SYSTEM CODEC_TESTL (* PUBL/SUBL Test *)
  (* Standard: 61499 Feasibility Demo *)
  (* Version 0.0, 2001-10-04, JHC, Rockwell Automation, Copied/modified from CODEC_TEST *)
  APPLICATION TEST_BITS (* Test bit string data types *)
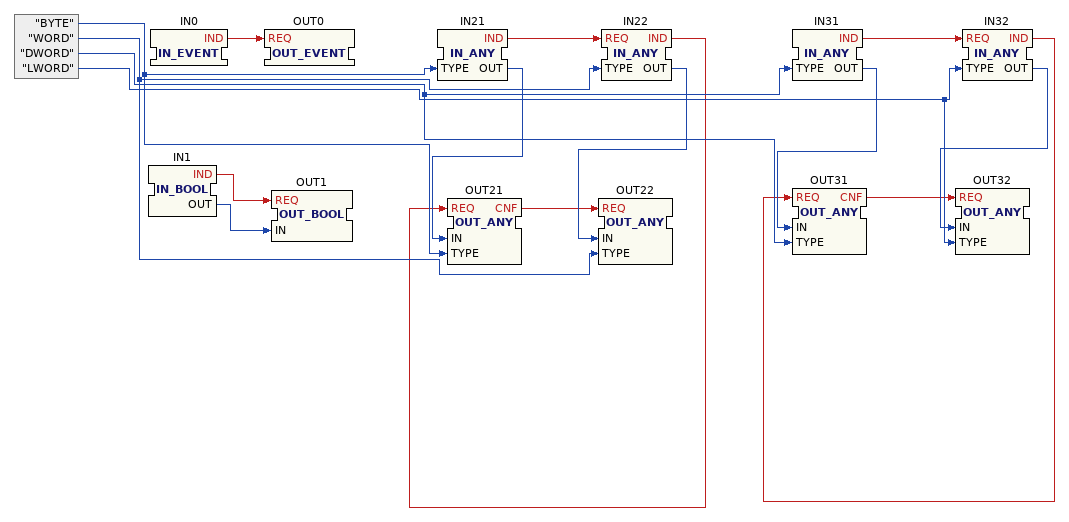
    FBS
      IN0 : IN_EVENT;
      OUT0 : OUT_EVENT;
      IN1 : IN_BOOL;
      OUT1 : OUT_BOOL;
      IN21 : IN_ANY;
      OUT21 : OUT_ANY;
      IN22 : IN_ANY;
      OUT22 : OUT_ANY;
      IN31 : IN_ANY;
      OUT31 : OUT_ANY;
      IN32 : IN_ANY;
      OUT32 : OUT_ANY;
    END_FBS
    EVENT_CONNECTIONS
      IN0.IND TO OUT0.REQ;
      IN1.IND TO OUT1.REQ;
      IN21.IND TO IN22.REQ;
      IN22.IND TO OUT21.REQ;
      OUT21.CNF TO OUT22.REQ;
      IN31.IND TO IN32.REQ;
      IN32.IND TO OUT31.REQ;
      OUT31.CNF TO OUT32.REQ;
    END_CONNECTIONS
    DATA_CONNECTIONS
      IN1.OUT TO OUT1.IN;
      IN21.OUT TO OUT21.IN;
      IN22.OUT TO OUT22.IN;
      IN31.OUT TO OUT31.IN;
      IN32.OUT TO OUT32.IN;
      "BYTE" TO IN21.TYPE;
      "BYTE" TO OUT21.TYPE;
      "WORD" TO IN22.TYPE;
      "WORD" TO OUT22.TYPE;
      "DWORD" TO IN31.TYPE;
      "DWORD" TO OUT31.TYPE;
      "LWORD" TO IN32.TYPE;
      "LWORD" TO OUT32.TYPE;
    END_CONNECTIONS
  END_APPLICATION
  APPLICATION TEST_INTS (* Test integer data types *)
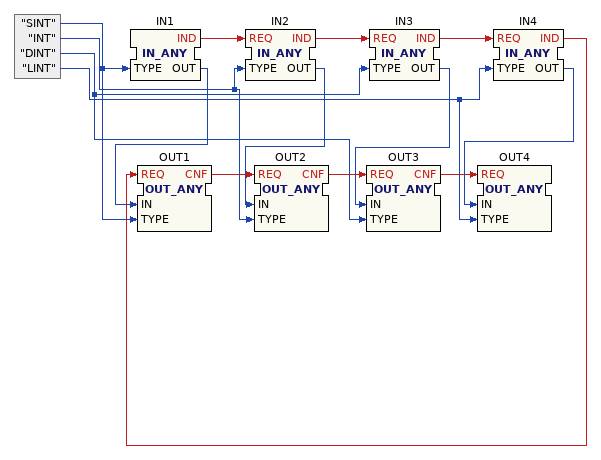
    FBS
      IN1 : IN_ANY;
      IN2 : IN_ANY;
      IN3 : IN_ANY;
      IN4 : IN_ANY;
      OUT1 : OUT_ANY;
      OUT2 : OUT_ANY;
      OUT3 : OUT_ANY;
      OUT4 : OUT_ANY;
    END_FBS
    EVENT_CONNECTIONS
      IN1.IND TO IN2.REQ;
      IN2.IND TO IN3.REQ;
      IN3.IND TO IN4.REQ;
      IN4.IND TO OUT1.REQ;
      OUT1.CNF TO OUT2.REQ;
      OUT2.CNF TO OUT3.REQ;
      OUT3.CNF TO OUT4.REQ;
    END_CONNECTIONS
    DATA_CONNECTIONS
      IN1.OUT TO OUT1.IN;
      IN2.OUT TO OUT2.IN;
      IN3.OUT TO OUT3.IN;
      IN4.OUT TO OUT4.IN;
      "SINT" TO IN1.TYPE;
      "SINT" TO OUT1.TYPE;
      "INT" TO IN2.TYPE;
      "INT" TO OUT2.TYPE;
      "DINT" TO IN3.TYPE;
      "DINT" TO OUT3.TYPE;
      "LINT" TO IN4.TYPE;
      "LINT" TO OUT4.TYPE;
    END_CONNECTIONS
  END_APPLICATION
  APPLICATION TEST_UINTS (* Test unsigned integer data types *)
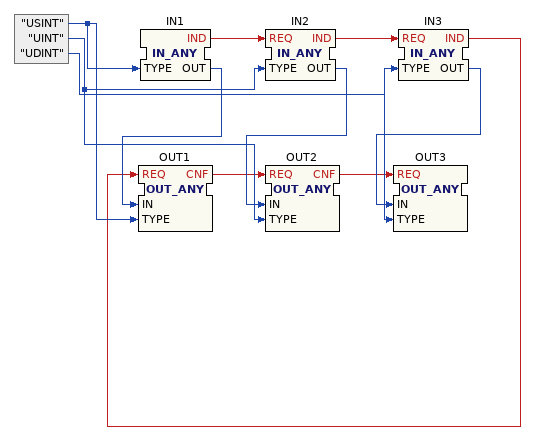
    FBS
      IN1 : IN_ANY;
      IN2 : IN_ANY;
      IN3 : IN_ANY;
      OUT1 : OUT_ANY;
      OUT2 : OUT_ANY;
      OUT3 : OUT_ANY;
    END_FBS
    EVENT_CONNECTIONS
      IN1.IND TO IN2.REQ;
      IN2.IND TO IN3.REQ;
      IN3.IND TO OUT1.REQ;
      OUT1.CNF TO OUT2.REQ;
      OUT2.CNF TO OUT3.REQ;
    END_CONNECTIONS
    DATA_CONNECTIONS
      IN1.OUT TO OUT1.IN;
      IN2.OUT TO OUT2.IN;
      IN3.OUT TO OUT3.IN;
      "USINT" TO IN1.TYPE;
      "USINT" TO OUT1.TYPE;
      "UINT" TO IN2.TYPE;
      "UINT" TO OUT2.TYPE;
      "UDINT" TO IN3.TYPE;
      "UDINT" TO OUT3.TYPE;
    END_CONNECTIONS
  END_APPLICATION
  APPLICATION TEST_REALS (* Test floating point data types *)
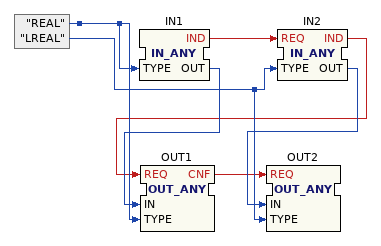
    FBS
      IN1 : IN_ANY;
      IN2 : IN_ANY;
      OUT1 : OUT_ANY;
      OUT2 : OUT_ANY;
    END_FBS
    EVENT_CONNECTIONS
      IN1.IND TO IN2.REQ;
      IN2.IND TO OUT1.REQ;
      OUT1.CNF TO OUT2.REQ;
    END_CONNECTIONS
    DATA_CONNECTIONS
      IN1.OUT TO OUT1.IN;
      IN2.OUT TO OUT2.IN;
      "REAL" TO IN1.TYPE;
      "REAL" TO OUT1.TYPE;
      "LREAL" TO IN2.TYPE;
      "LREAL" TO OUT2.TYPE;
    END_CONNECTIONS
  END_APPLICATION
  APPLICATION TEST_TIMES (* Test time data types *)
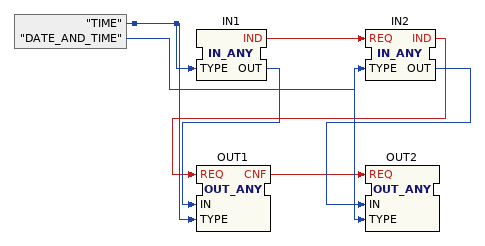
    FBS
      IN1 : IN_ANY;
      IN2 : IN_ANY;
      OUT1 : OUT_ANY;
      OUT2 : OUT_ANY;
    END_FBS
    EVENT_CONNECTIONS
      IN1.IND TO IN2.REQ;
      IN2.IND TO OUT1.REQ;
      OUT1.CNF TO OUT2.REQ;
    END_CONNECTIONS
    DATA_CONNECTIONS
      IN1.OUT TO OUT1.IN;
      IN2.OUT TO OUT2.IN;
      "TIME" TO IN1.TYPE;
      "TIME" TO OUT1.TYPE;
      "DATE_AND_TIME" TO IN2.TYPE;
      "DATE_AND_TIME" TO OUT2.TYPE;
    END_CONNECTIONS
  END_APPLICATION
  APPLICATION TEST_STRINGS (* Test string data types *)
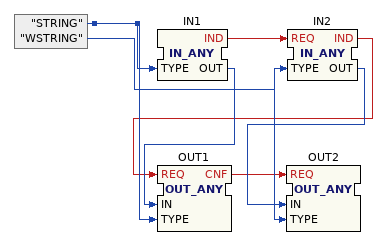
    FBS
      IN1 : IN_ANY;
      IN2 : IN_ANY;
      OUT1 : OUT_ANY;
      OUT2 : OUT_ANY;
    END_FBS
    EVENT_CONNECTIONS
      IN1.IND TO IN2.REQ;
      IN2.IND TO OUT1.REQ;
      OUT1.CNF TO OUT2.REQ;
    END_CONNECTIONS
    DATA_CONNECTIONS
      IN1.OUT TO OUT1.IN;
      IN2.OUT TO OUT2.IN;
      "STRING" TO IN1.TYPE;
      "STRING" TO OUT1.TYPE;
      "WSTRING" TO IN2.TYPE;
      "WSTRING" TO OUT2.TYPE;
    END_CONNECTIONS
  END_APPLICATION
  APPLICATION TEST_ARRAY (* Test ARRAYs *)
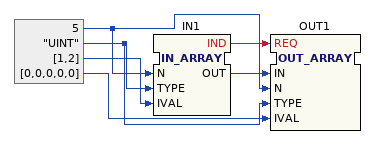
    FBS
      IN1 : IN_ARRAY;
      OUT1 : OUT_ARRAY;
    END_FBS
    EVENT_CONNECTIONS
      IN1.IND TO OUT1.REQ;
    END_CONNECTIONS
    DATA_CONNECTIONS
      IN1.OUT TO OUT1.IN;
      5 TO IN1.N;
      5 TO OUT1.N;
      "UINT" TO IN1.TYPE;
      "UINT" TO OUT1.TYPE;
      [1,2] TO IN1.IVAL;
      [0,0,0,0,0] TO OUT1.IVAL;
    END_CONNECTIONS
  END_APPLICATION
  APPLICATION TEST_COLOR (* Test  COLOR - Just for fun! *)
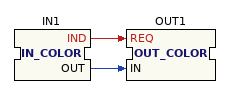
    FBS
      IN1 : IN_COLOR;
      OUT1 : OUT_COLOR;
    END_FBS
    EVENT_CONNECTIONS
      IN1.IND TO OUT1.REQ;
    END_CONNECTIONS
    DATA_CONNECTIONS
      IN1.OUT TO OUT1.IN;
    END_CONNECTIONS
  END_APPLICATION
  DEVICE SEND_BITS : FRAME_DEVICE
    RESOURCE RES0 : PANEL_RESOURCE
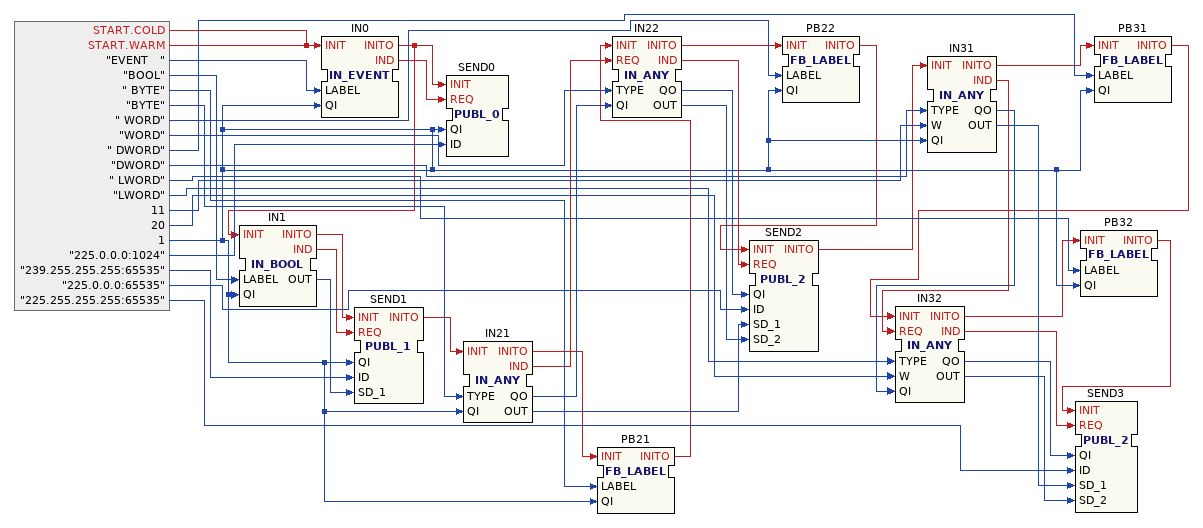
      FBS
        IN0 : IN_EVENT;
        SEND0 : PUBL_0;
        IN1 : IN_BOOL;
        SEND1 : PUBL_1;
        PB21 : FB_LABEL;
        IN21 : IN_ANY;
        PB22 : FB_LABEL;
        IN22 : IN_ANY;
        SEND2 : PUBL_2;
        PB31 : FB_LABEL;
        IN31 : IN_ANY;
        PB32 : FB_LABEL;
        IN32 : IN_ANY;
        SEND3 : PUBL_2;
      END_FBS
      EVENT_CONNECTIONS
        START.COLD TO IN0.INIT;
        START.WARM TO IN0.INIT;
        IN0.INITO TO SEND0.INIT;
        IN0.INITO TO IN1.INIT;
        IN1.INITO TO SEND1.INIT;
        SEND1.INITO TO IN21.INIT;
        IN21.INITO TO PB21.INIT;
        PB21.INITO TO IN22.INIT;
        IN22.INITO TO PB22.INIT;
        PB22.INITO TO SEND2.INIT;
        SEND2.INITO TO IN31.INIT;
        IN31.INITO TO PB31.INIT;
        PB31.INITO TO IN32.INIT;
        IN32.INITO TO PB32.INIT;
        PB32.INITO TO SEND3.INIT;
        IN0.IND TO SEND0.REQ;
        IN1.IND TO SEND1.REQ;
        IN21.IND TO IN22.REQ;
        IN22.IND TO SEND2.REQ;
        IN31.IND TO IN32.REQ;
        IN32.IND TO SEND3.REQ;
      END_CONNECTIONS
      DATA_CONNECTIONS
        "EVENT   " TO IN0.LABEL;
        "BOOL" TO IN1.LABEL;
        " BYTE" TO PB21.LABEL;
        "BYTE" TO IN21.TYPE;
        " WORD" TO PB22.LABEL;
        "WORD" TO IN22.TYPE;
        " DWORD" TO PB31.LABEL;
        "DWORD" TO IN31.TYPE;
        " LWORD" TO PB32.LABEL;
        "LWORD" TO IN32.TYPE;
        11 TO IN31.W;
        20 TO IN32.W;
        1 TO IN0.QI;
        1 TO IN1.QI;
        1 TO SEND0.QI;
        1 TO SEND1.QI;
        1 TO IN21.QI;
        IN21.QO TO IN22.QI;
        1 TO PB21.QI;
        1 TO PB22.QI;
        IN22.QO TO SEND2.QI;
        1 TO IN31.QI;
        IN31.QO TO IN32.QI;
        1 TO PB31.QI;
        1 TO PB32.QI;
        IN32.QO TO SEND3.QI;
        "225.0.0.0:1024" TO SEND0.ID;
        "239.255.255.255:65535" TO SEND1.ID;
        "225.0.0.0:65535" TO SEND2.ID;
        "225.255.255.255:65535" TO SEND3.ID;
        IN1.OUT TO SEND1.SD_1;
        IN21.OUT TO SEND2.SD_1;
        IN22.OUT TO SEND2.SD_2;
        IN31.OUT TO SEND3.SD_1;
        IN32.OUT TO SEND3.SD_2;
      END_CONNECTIONS
    END_RESOURCE
  END_DEVICE
  DEVICE RCV_BITS : FRAME_DEVICE
    RESOURCE RES0 : PANEL_RESOURCE
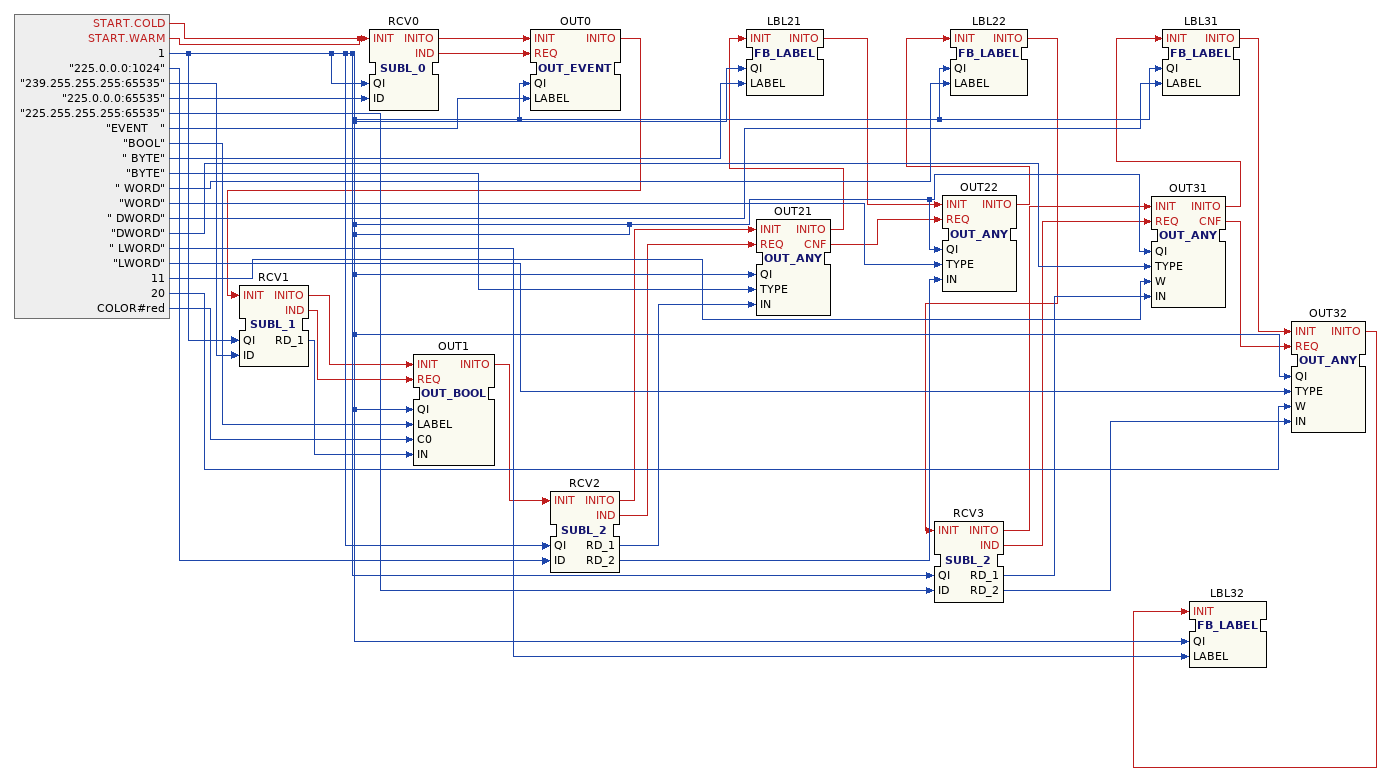
      FBS
        RCV0 : SUBL_0;
        OUT0 : OUT_EVENT;
        RCV1 : SUBL_1;
        OUT1 : OUT_BOOL;
        RCV2 : SUBL_2;
        LBL21 : FB_LABEL;
        OUT21 : OUT_ANY;
        LBL22 : FB_LABEL;
        OUT22 : OUT_ANY;
        RCV3 : SUBL_2;
        LBL31 : FB_LABEL;
        OUT31 : OUT_ANY;
        LBL32 : FB_LABEL;
        OUT32 : OUT_ANY;
      END_FBS
      EVENT_CONNECTIONS
        START.COLD TO RCV0.INIT;
        START.WARM TO RCV0.INIT;
        RCV0.INITO TO OUT0.INIT;
        OUT0.INITO TO RCV1.INIT;
        RCV1.INITO TO OUT1.INIT;
        OUT1.INITO TO RCV2.INIT;
        RCV2.INITO TO OUT21.INIT;
        OUT21.INITO TO LBL21.INIT;
        LBL21.INITO TO OUT22.INIT;
        OUT22.INITO TO LBL22.INIT;
        LBL22.INITO TO RCV3.INIT;
        RCV3.INITO TO OUT31.INIT;
        OUT31.INITO TO LBL31.INIT;
        LBL31.INITO TO OUT32.INIT;
        OUT32.INITO TO LBL32.INIT;
        RCV0.IND TO OUT0.REQ;
        RCV1.IND TO OUT1.REQ;
        RCV2.IND TO OUT21.REQ;
        OUT21.CNF TO OUT22.REQ;
        RCV3.IND TO OUT31.REQ;
        OUT31.CNF TO OUT32.REQ;
      END_CONNECTIONS
      DATA_CONNECTIONS
        1 TO RCV0.QI;
        1 TO RCV1.QI;
        1 TO RCV2.QI;
        1 TO RCV3.QI;
        "225.0.0.0:1024" TO RCV0.ID;
        "239.255.255.255:65535" TO RCV1.ID;
        "225.0.0.0:65535" TO RCV2.ID;
        "225.255.255.255:65535" TO RCV3.ID;
        1 TO OUT0.QI;
        1 TO OUT1.QI;
        1 TO OUT21.QI;
        1 TO OUT22.QI;
        1 TO LBL21.QI;
        1 TO LBL22.QI;
        1 TO OUT31.QI;
        1 TO OUT32.QI;
        1 TO LBL31.QI;
        1 TO LBL32.QI;
        "EVENT   " TO OUT0.LABEL;
        "BOOL" TO OUT1.LABEL;
        " BYTE" TO LBL21.LABEL;
        "BYTE" TO OUT21.TYPE;
        " WORD" TO LBL22.LABEL;
        "WORD" TO OUT22.TYPE;
        " DWORD" TO LBL31.LABEL;
        "DWORD" TO OUT31.TYPE;
        " LWORD" TO LBL32.LABEL;
        "LWORD" TO OUT32.TYPE;
        11 TO OUT31.W;
        20 TO OUT32.W;
        COLOR#red TO OUT1.C0;
        RCV1.RD_1 TO OUT1.IN;
        RCV2.RD_1 TO OUT21.IN;
        RCV2.RD_2 TO OUT22.IN;
        RCV3.RD_1 TO OUT31.IN;
        RCV3.RD_2 TO OUT32.IN;
      END_CONNECTIONS
    END_RESOURCE
    DATA_CONNECTIONS
      0 TO RES0.TRACE;
    END_CONNECTIONS
  END_DEVICE
  DEVICE SEND_INTS : FRAME_DEVICE
    RESOURCE RES0 : PANEL_RESOURCE
      FBS
        PB1 : FB_LABEL;
        IN1 : IN_ANY;
        PB2 : FB_LABEL;
        IN2 : IN_ANY;
        PB3 : FB_LABEL;
        IN3 : IN_ANY;
        PB4 : FB_LABEL;
        IN4 : IN_ANY;
        SEND : PUBL_4;
      END_FBS
      EVENT_CONNECTIONS
        START.COLD TO IN1.INIT;
        START.WARM TO IN1.INIT;
        IN1.INITO TO PB1.INIT;
        PB1.INITO TO IN2.INIT;
        IN2.INITO TO PB2.INIT;
        PB2.INITO TO IN3.INIT;
        IN3.INITO TO PB3.INIT;
        PB3.INITO TO IN4.INIT;
        IN4.INITO TO PB4.INIT;
        PB4.INITO TO SEND.INIT;
        IN1.IND TO IN2.REQ;
        IN2.IND TO IN3.REQ;
        IN3.IND TO IN4.REQ;
        IN4.IND TO SEND.REQ;
      END_CONNECTIONS
      DATA_CONNECTIONS
        " SINT" TO PB1.LABEL;
        " INT" TO PB2.LABEL;
        " DINT" TO PB3.LABEL;
        " LINT" TO PB4.LABEL;
        "SINT" TO IN1.TYPE;
        "INT" TO IN2.TYPE;
        "DINT" TO IN3.TYPE;
        "LINT" TO IN4.TYPE;
        11 TO IN3.W;
        20 TO IN4.W;
        1 TO IN1.QI;
        IN1.QO TO IN2.QI;
        1 TO PB1.QI;
        1 TO PB2.QI;
        IN2.QO TO IN3.QI;
        IN3.QO TO IN4.QI;
        1 TO PB3.QI;
        1 TO PB4.QI;
        IN4.QO TO SEND.QI;
        "239.0.0.1:1024" TO SEND.ID;
        IN1.OUT TO SEND.SD_1;
        IN2.OUT TO SEND.SD_2;
        IN3.OUT TO SEND.SD_3;
        IN4.OUT TO SEND.SD_4;
      END_CONNECTIONS
    END_RESOURCE
  END_DEVICE
  DEVICE RCV_INTS : FRAME_DEVICE
    RESOURCE RES0 : PANEL_RESOURCE
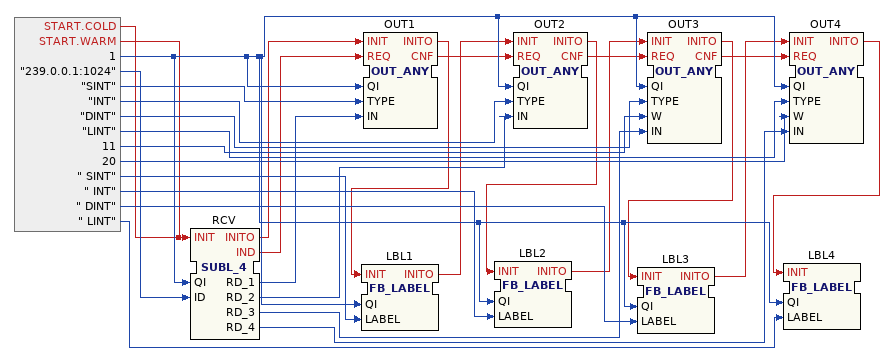
      FBS
        RCV : SUBL_4;
        LBL1 : FB_LABEL;
        OUT1 : OUT_ANY;
        LBL2 : FB_LABEL;
        OUT2 : OUT_ANY;
        LBL3 : FB_LABEL;
        OUT3 : OUT_ANY;
        LBL4 : FB_LABEL;
        OUT4 : OUT_ANY;
      END_FBS
      EVENT_CONNECTIONS
        START.COLD TO RCV.INIT;
        START.WARM TO RCV.INIT;
        RCV.INITO TO OUT1.INIT;
        OUT1.INITO TO LBL1.INIT;
        LBL1.INITO TO OUT2.INIT;
        OUT2.INITO TO LBL2.INIT;
        LBL2.INITO TO OUT3.INIT;
        OUT3.INITO TO LBL3.INIT;
        LBL3.INITO TO OUT4.INIT;
        OUT4.INITO TO LBL4.INIT;
        RCV.IND TO OUT1.REQ;
        OUT1.CNF TO OUT2.REQ;
        OUT2.CNF TO OUT3.REQ;
        OUT3.CNF TO OUT4.REQ;
      END_CONNECTIONS
      DATA_CONNECTIONS
        1 TO RCV.QI;
        "239.0.0.1:1024" TO RCV.ID;
        1 TO OUT1.QI;
        1 TO OUT2.QI;
        1 TO LBL1.QI;
        1 TO LBL2.QI;
        1 TO OUT3.QI;
        1 TO OUT4.QI;
        1 TO LBL3.QI;
        1 TO LBL4.QI;
        "SINT" TO OUT1.TYPE;
        "INT" TO OUT2.TYPE;
        "DINT" TO OUT3.TYPE;
        "LINT" TO OUT4.TYPE;
        11 TO OUT3.W;
        20 TO OUT4.W;
        " SINT" TO LBL1.LABEL;
        " INT" TO LBL2.LABEL;
        " DINT" TO LBL3.LABEL;
        " LINT" TO LBL4.LABEL;
        RCV.RD_1 TO OUT1.IN;
        RCV.RD_2 TO OUT2.IN;
        RCV.RD_3 TO OUT3.IN;
        RCV.RD_4 TO OUT4.IN;
      END_CONNECTIONS
    END_RESOURCE
    DATA_CONNECTIONS
      0 TO RES0.TRACE;
    END_CONNECTIONS
  END_DEVICE
  DEVICE SEND_UINTS : FRAME_DEVICE
    RESOURCE RES0 : PANEL_RESOURCE
      FBS
        PB1 : FB_LABEL;
        IN1 : IN_ANY;
        PB2 : FB_LABEL;
        IN2 : IN_ANY;
        PB3 : FB_LABEL;
        IN3 : IN_ANY;
        SEND : PUBL_3;
      END_FBS
      EVENT_CONNECTIONS
        START.COLD TO IN1.INIT;
        START.WARM TO IN1.INIT;
        IN1.INITO TO PB1.INIT;
        PB1.INITO TO IN2.INIT;
        IN2.INITO TO PB2.INIT;
        PB2.INITO TO IN3.INIT;
        IN3.INITO TO PB3.INIT;
        PB3.INITO TO SEND.INIT;
        IN1.IND TO IN2.REQ;
        IN2.IND TO IN3.REQ;
        IN3.IND TO SEND.REQ;
      END_CONNECTIONS
      DATA_CONNECTIONS
        " USINT" TO PB1.LABEL;
        " UINT" TO PB2.LABEL;
        " UDINT" TO PB3.LABEL;
        "USINT" TO IN1.TYPE;
        "UINT" TO IN2.TYPE;
        "UDINT" TO IN3.TYPE;
        11 TO IN3.W;
        1 TO IN1.QI;
        IN1.QO TO IN2.QI;
        1 TO PB1.QI;
        1 TO PB2.QI;
        IN2.QO TO IN3.QI;
        1 TO PB3.QI;
        IN3.QO TO SEND.QI;
        "239.0.0.1:65535" TO SEND.ID;
        IN1.OUT TO SEND.SD_1;
        IN2.OUT TO SEND.SD_2;
        IN3.OUT TO SEND.SD_3;
      END_CONNECTIONS
    END_RESOURCE
  END_DEVICE
  DEVICE RCV_UINTS : FRAME_DEVICE
    RESOURCE RES0 : PANEL_RESOURCE
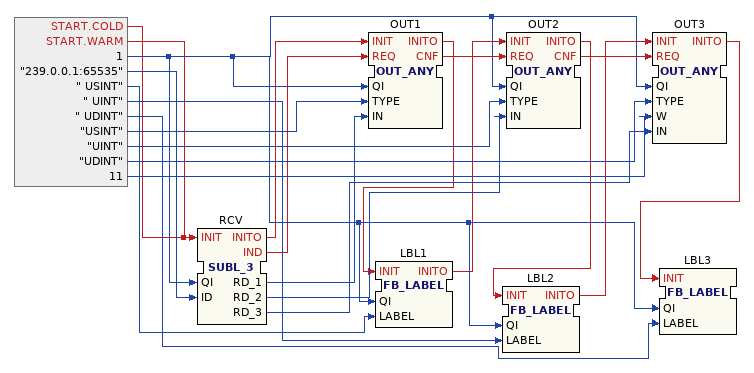
      FBS
        RCV : SUBL_3;
        LBL1 : FB_LABEL;
        OUT1 : OUT_ANY;
        LBL2 : FB_LABEL;
        OUT2 : OUT_ANY;
        LBL3 : FB_LABEL;
        OUT3 : OUT_ANY;
      END_FBS
      EVENT_CONNECTIONS
        START.COLD TO RCV.INIT;
        START.WARM TO RCV.INIT;
        RCV.INITO TO OUT1.INIT;
        OUT1.INITO TO LBL1.INIT;
        LBL1.INITO TO OUT2.INIT;
        OUT2.INITO TO LBL2.INIT;
        LBL2.INITO TO OUT3.INIT;
        OUT3.INITO TO LBL3.INIT;
        RCV.IND TO OUT1.REQ;
        OUT1.CNF TO OUT2.REQ;
        OUT2.CNF TO OUT3.REQ;
      END_CONNECTIONS
      DATA_CONNECTIONS
        1 TO RCV.QI;
        "239.0.0.1:65535" TO RCV.ID;
        1 TO OUT1.QI;
        1 TO OUT2.QI;
        1 TO LBL1.QI;
        1 TO LBL2.QI;
        1 TO OUT3.QI;
        1 TO LBL3.QI;
        " USINT" TO LBL1.LABEL;
        " UINT" TO LBL2.LABEL;
        " UDINT" TO LBL3.LABEL;
        "USINT" TO OUT1.TYPE;
        "UINT" TO OUT2.TYPE;
        "UDINT" TO OUT3.TYPE;
        11 TO OUT3.W;
        RCV.RD_1 TO OUT1.IN;
        RCV.RD_2 TO OUT2.IN;
        RCV.RD_3 TO OUT3.IN;
      END_CONNECTIONS
    END_RESOURCE
    DATA_CONNECTIONS
      0 TO RES0.TRACE;
    END_CONNECTIONS
  END_DEVICE
  DEVICE SEND_REALS : FRAME_DEVICE
    RESOURCE RES0 : PANEL_RESOURCE
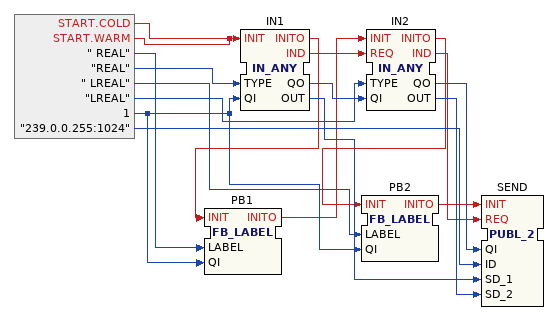
      FBS
        PB1 : FB_LABEL;
        IN1 : IN_ANY;
        PB2 : FB_LABEL;
        IN2 : IN_ANY;
        SEND : PUBL_2;
      END_FBS
      EVENT_CONNECTIONS
        START.COLD TO IN1.INIT;
        START.WARM TO IN1.INIT;
        IN1.INITO TO PB1.INIT;
        PB1.INITO TO IN2.INIT;
        IN2.INITO TO PB2.INIT;
        PB2.INITO TO SEND.INIT;
        IN1.IND TO IN2.REQ;
        IN2.IND TO SEND.REQ;
      END_CONNECTIONS
      DATA_CONNECTIONS
        " REAL" TO PB1.LABEL;
        "REAL" TO IN1.TYPE;
        " LREAL" TO PB2.LABEL;
        "LREAL" TO IN2.TYPE;
        1 TO IN1.QI;
        IN1.QO TO IN2.QI;
        1 TO PB1.QI;
        1 TO PB2.QI;
        IN2.QO TO SEND.QI;
        "239.0.0.255:1024" TO SEND.ID;
        IN1.OUT TO SEND.SD_1;
        IN2.OUT TO SEND.SD_2;
      END_CONNECTIONS
    END_RESOURCE
  END_DEVICE
  DEVICE RCV_REALS : FRAME_DEVICE
    RESOURCE RES0 : PANEL_RESOURCE
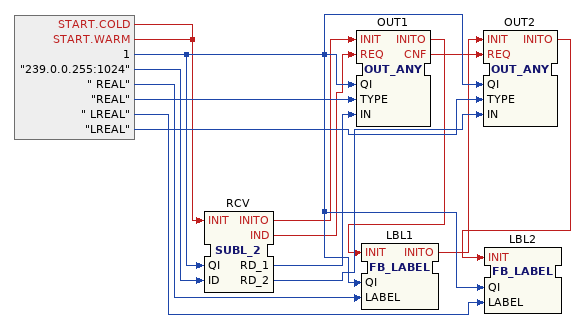
      FBS
        RCV : SUBL_2;
        LBL1 : FB_LABEL;
        OUT1 : OUT_ANY;
        LBL2 : FB_LABEL;
        OUT2 : OUT_ANY;
      END_FBS
      EVENT_CONNECTIONS
        START.COLD TO RCV.INIT;
        START.WARM TO RCV.INIT;
        RCV.INITO TO OUT1.INIT;
        OUT1.INITO TO LBL1.INIT;
        LBL1.INITO TO OUT2.INIT;
        OUT2.INITO TO LBL2.INIT;
        RCV.IND TO OUT1.REQ;
        OUT1.CNF TO OUT2.REQ;
      END_CONNECTIONS
      DATA_CONNECTIONS
        1 TO RCV.QI;
        "239.0.0.255:1024" TO RCV.ID;
        1 TO OUT1.QI;
        1 TO OUT2.QI;
        1 TO LBL1.QI;
        1 TO LBL2.QI;
        " REAL" TO LBL1.LABEL;
        "REAL" TO OUT1.TYPE;
        " LREAL" TO LBL2.LABEL;
        "LREAL" TO OUT2.TYPE;
        RCV.RD_1 TO OUT1.IN;
        RCV.RD_2 TO OUT2.IN;
      END_CONNECTIONS
    END_RESOURCE
    DATA_CONNECTIONS
      0 TO RES0.TRACE;
    END_CONNECTIONS
  END_DEVICE
  DEVICE SEND_TIMES : FRAME_DEVICE
    RESOURCE RES0 : PANEL_RESOURCE
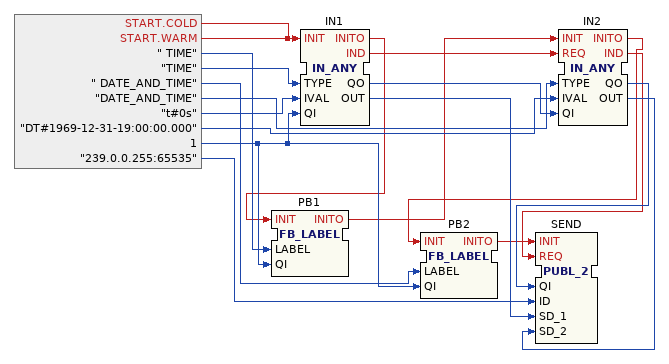
      FBS
        PB1 : FB_LABEL;
        IN1 : IN_ANY;
        PB2 : FB_LABEL;
        IN2 : IN_ANY;
        SEND : PUBL_2;
      END_FBS
      EVENT_CONNECTIONS
        START.COLD TO IN1.INIT;
        START.WARM TO IN1.INIT;
        IN1.INITO TO PB1.INIT;
        PB1.INITO TO IN2.INIT;
        IN2.INITO TO PB2.INIT;
        PB2.INITO TO SEND.INIT;
        IN1.IND TO IN2.REQ;
        IN2.IND TO SEND.REQ;
      END_CONNECTIONS
      DATA_CONNECTIONS
        " TIME" TO PB1.LABEL;
        "TIME" TO IN1.TYPE;
        " DATE_AND_TIME" TO PB2.LABEL;
        "DATE_AND_TIME" TO IN2.TYPE;
        "t#0s" TO IN1.IVAL;
        "DT#1969-12-31-19:00:00.000" TO IN2.IVAL;
        1 TO IN1.QI;
        IN1.QO TO IN2.QI;
        1 TO PB1.QI;
        1 TO PB2.QI;
        IN2.QO TO SEND.QI;
        "239.0.0.255:65535" TO SEND.ID;
        IN1.OUT TO SEND.SD_1;
        IN2.OUT TO SEND.SD_2;
      END_CONNECTIONS
    END_RESOURCE
  END_DEVICE
  DEVICE RCV_TIMES : FRAME_DEVICE
    RESOURCE RES0 : PANEL_RESOURCE
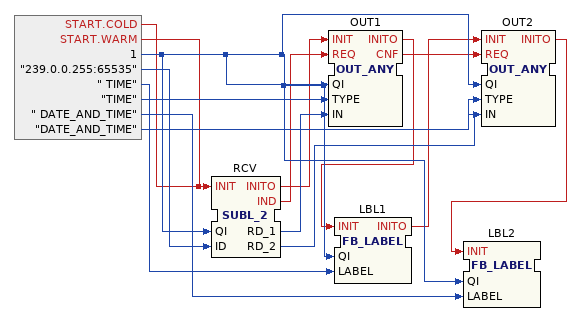
      FBS
        RCV : SUBL_2;
        LBL1 : FB_LABEL;
        OUT1 : OUT_ANY;
        LBL2 : FB_LABEL;
        OUT2 : OUT_ANY;
      END_FBS
      EVENT_CONNECTIONS
        START.COLD TO RCV.INIT;
        START.WARM TO RCV.INIT;
        RCV.INITO TO OUT1.INIT;
        OUT1.INITO TO LBL1.INIT;
        LBL1.INITO TO OUT2.INIT;
        OUT2.INITO TO LBL2.INIT;
        RCV.IND TO OUT1.REQ;
        OUT1.CNF TO OUT2.REQ;
      END_CONNECTIONS
      DATA_CONNECTIONS
        1 TO RCV.QI;
        "239.0.0.255:65535" TO RCV.ID;
        1 TO OUT1.QI;
        1 TO OUT2.QI;
        1 TO LBL1.QI;
        1 TO LBL2.QI;
        " TIME" TO LBL1.LABEL;
        "TIME" TO OUT1.TYPE;
        " DATE_AND_TIME" TO LBL2.LABEL;
        "DATE_AND_TIME" TO OUT2.TYPE;
        RCV.RD_1 TO OUT1.IN;
        RCV.RD_2 TO OUT2.IN;
      END_CONNECTIONS
    END_RESOURCE
    DATA_CONNECTIONS
      0 TO RES0.TRACE;
    END_CONNECTIONS
  END_DEVICE
  DEVICE SEND_STRINGS : FRAME_DEVICE
    RESOURCE RES0 : PANEL_RESOURCE
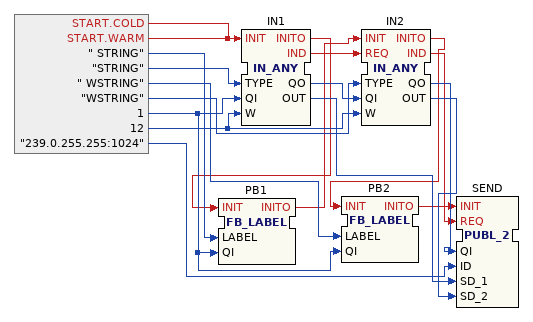
      FBS
        PB1 : FB_LABEL;
        IN1 : IN_ANY;
        PB2 : FB_LABEL;
        IN2 : IN_ANY;
        SEND : PUBL_2;
      END_FBS
      EVENT_CONNECTIONS
        START.COLD TO IN1.INIT;
        START.WARM TO IN1.INIT;
        IN1.INITO TO PB1.INIT;
        PB1.INITO TO IN2.INIT;
        IN2.INITO TO PB2.INIT;
        PB2.INITO TO SEND.INIT;
        IN1.IND TO IN2.REQ;
        IN2.IND TO SEND.REQ;
      END_CONNECTIONS
      DATA_CONNECTIONS
        " STRING" TO PB1.LABEL;
        "STRING" TO IN1.TYPE;
        " WSTRING" TO PB2.LABEL;
        "WSTRING" TO IN2.TYPE;
        1 TO IN1.QI;
        IN1.QO TO IN2.QI;
        1 TO PB1.QI;
        1 TO PB2.QI;
        IN2.QO TO SEND.QI;
        12 TO IN1.W;
        12 TO IN2.W;
        "239.0.255.255:1024" TO SEND.ID;
        IN1.OUT TO SEND.SD_1;
        IN2.OUT TO SEND.SD_2;
      END_CONNECTIONS
    END_RESOURCE
  END_DEVICE
  DEVICE RCV_STRINGS : FRAME_DEVICE
    RESOURCE RES0 : PANEL_RESOURCE
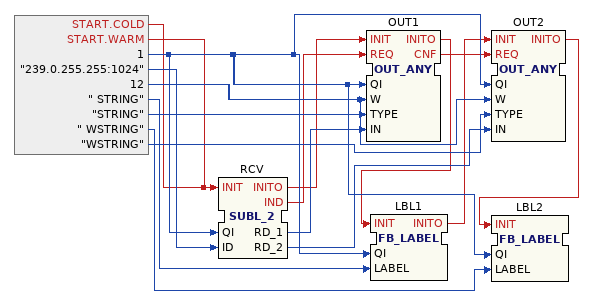
      FBS
        RCV : SUBL_2;
        LBL1 : FB_LABEL;
        OUT1 : OUT_ANY;
        LBL2 : FB_LABEL;
        OUT2 : OUT_ANY;
      END_FBS
      EVENT_CONNECTIONS
        START.COLD TO RCV.INIT;
        START.WARM TO RCV.INIT;
        RCV.INITO TO OUT1.INIT;
        OUT1.INITO TO LBL1.INIT;
        LBL1.INITO TO OUT2.INIT;
        OUT2.INITO TO LBL2.INIT;
        RCV.IND TO OUT1.REQ;
        OUT1.CNF TO OUT2.REQ;
      END_CONNECTIONS
      DATA_CONNECTIONS
        1 TO RCV.QI;
        "239.0.255.255:1024" TO RCV.ID;
        1 TO OUT1.QI;
        1 TO OUT2.QI;
        1 TO LBL1.QI;
        1 TO LBL2.QI;
        12 TO OUT1.W;
        12 TO OUT2.W;
        " STRING" TO LBL1.LABEL;
        "STRING" TO OUT1.TYPE;
        " WSTRING" TO LBL2.LABEL;
        "WSTRING" TO OUT2.TYPE;
        RCV.RD_1 TO OUT1.IN;
        RCV.RD_2 TO OUT2.IN;
      END_CONNECTIONS
    END_RESOURCE
    DATA_CONNECTIONS
      0 TO RES0.TRACE;
    END_CONNECTIONS
  END_DEVICE
  DEVICE SEND_ARRAY : FRAME_DEVICE
    RESOURCE RES0 : PANEL_RESOURCE
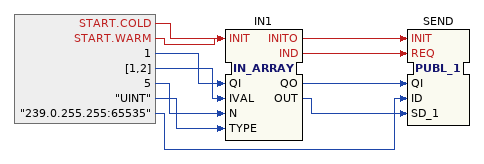
      FBS
        IN1 : IN_ARRAY;
        SEND : PUBL_1;
      END_FBS
      EVENT_CONNECTIONS
        START.COLD TO IN1.INIT;
        START.WARM TO IN1.INIT;
        IN1.INITO TO SEND.INIT;
        IN1.IND TO SEND.REQ;
      END_CONNECTIONS
      DATA_CONNECTIONS
        1 TO IN1.QI;
        IN1.QO TO SEND.QI;
        [1,2] TO IN1.IVAL;
        5 TO IN1.N;
        "UINT" TO IN1.TYPE;
        "239.0.255.255:65535" TO SEND.ID;
        IN1.OUT TO SEND.SD_1;
      END_CONNECTIONS
    END_RESOURCE
  END_DEVICE
  DEVICE RCV_ARRAY : FRAME_DEVICE
    RESOURCE RES0 : PANEL_RESOURCE
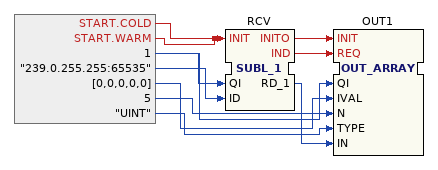
      FBS
        RCV : SUBL_1;
        OUT1 : OUT_ARRAY;
      END_FBS
      EVENT_CONNECTIONS
        START.COLD TO RCV.INIT;
        START.WARM TO RCV.INIT;
        RCV.INITO TO OUT1.INIT;
        RCV.IND TO OUT1.REQ;
      END_CONNECTIONS
      DATA_CONNECTIONS
        1 TO RCV.QI;
        "239.0.255.255:65535" TO RCV.ID;
        1 TO OUT1.QI;
        [0,0,0,0,0] TO OUT1.IVAL;
        5 TO OUT1.N;
        "UINT" TO OUT1.TYPE;
        RCV.RD_1 TO OUT1.IN;
      END_CONNECTIONS
    END_RESOURCE
    DATA_CONNECTIONS
      0 TO RES0.TRACE;
    END_CONNECTIONS
  END_DEVICE
  DEVICE SEND_COLOR : FRAME_DEVICE
    RESOURCE RES0 : PANEL_RESOURCE
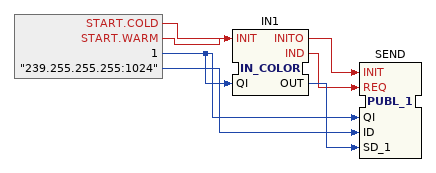
      FBS
        IN1 : IN_COLOR;
        SEND : PUBL_1;
      END_FBS
      EVENT_CONNECTIONS
        START.COLD TO IN1.INIT;
        START.WARM TO IN1.INIT;
        IN1.INITO TO SEND.INIT;
        IN1.IND TO SEND.REQ;
      END_CONNECTIONS
      DATA_CONNECTIONS
        1 TO IN1.QI;
        1 TO SEND.QI;
        "239.255.255.255:1024" TO SEND.ID;
        IN1.OUT TO SEND.SD_1;
      END_CONNECTIONS
    END_RESOURCE
  END_DEVICE
  DEVICE RCV_COLOR : FRAME_DEVICE
    RESOURCE RES0 : PANEL_RESOURCE
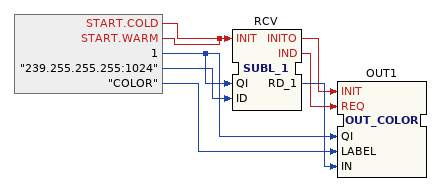
      FBS
        RCV : SUBL_1;
        OUT1 : OUT_COLOR;
      END_FBS
      EVENT_CONNECTIONS
        START.COLD TO RCV.INIT;
        START.WARM TO RCV.INIT;
        RCV.INITO TO OUT1.INIT;
        RCV.IND TO OUT1.REQ;
      END_CONNECTIONS
      DATA_CONNECTIONS
        1 TO RCV.QI;
        "239.255.255.255:1024" TO RCV.ID;
        1 TO OUT1.QI;
        "COLOR" TO OUT1.LABEL;
        RCV.RD_1 TO OUT1.IN;
      END_CONNECTIONS
    END_RESOURCE
    DATA_CONNECTIONS
      0 TO RES0.TRACE;
    END_CONNECTIONS
  END_DEVICE
  DATA_CONNECTIONS (* parameter values *)
    [50,50,175,195] TO SEND_BITS.BOUNDS;
    [225,50,175,195] TO RCV_BITS.BOUNDS;
    [50,240,175,170] TO SEND_INTS.BOUNDS;
    [225,240,175,170] TO RCV_INTS.BOUNDS;
    [50,405,175,120] TO SEND_UINTS.BOUNDS;
    [225,405,175,120] TO RCV_UINTS.BOUNDS;
    [50,520,175,90] TO SEND_REALS.BOUNDS;
    [225,520,175,90] TO RCV_REALS.BOUNDS;
    [400,240,200,120] TO SEND_TIMES.BOUNDS;
    [600,240,200,120] TO RCV_TIMES.BOUNDS;
    [400,355,200,95] TO SEND_STRINGS.BOUNDS;
    [600,355,200,95] TO RCV_STRINGS.BOUNDS;
    [400,445,210,70] TO SEND_ARRAY.BOUNDS;
    [610,445,190,70] TO RCV_ARRAY.BOUNDS;
    [400,510,210,70] TO SEND_COLOR.BOUNDS;
    [610,510,190,70] TO RCV_COLOR.BOUNDS;
    [1,1] TO SEND_BITS.GRID;
    [1,1] TO RCV_BITS.GRID;
    [1,1] TO SEND_INTS.GRID;
    [1,1] TO RCV_INTS.GRID;
    [1,1] TO SEND_UINTS.GRID;
    [1,1] TO RCV_UINTS.GRID;
    [1,1] TO SEND_REALS.GRID;
    [1,1] TO RCV_REALS.GRID;
    [1,1] TO SEND_TIMES.GRID;
    [1,1] TO RCV_TIMES.GRID;
    [1,1] TO SEND_STRINGS.GRID;
    [1,1] TO RCV_STRINGS.GRID;
    [1,1] TO SEND_ARRAY.GRID;
    [1,1] TO RCV_ARRAY.GRID;
    [1,1] TO SEND_COLOR.GRID;
    [1,1] TO RCV_COLOR.GRID;
  END_CONNECTIONS
  MAPPINGS
    TEST_BITS.IN0 ON SEND_BITS.RES0.IN0;
    TEST_BITS.OUT0 ON RCV_BITS.RES0.OUT0;
    TEST_BITS.IN1 ON SEND_BITS.RES0.IN1;
    TEST_BITS.OUT1 ON RCV_BITS.RES0.OUT1;
    TEST_BITS.PB21 ON SEND_BITS.RES0.PB21;
    TEST_BITS.IN21 ON SEND_BITS.RES0.IN21;
    TEST_BITS.PB22 ON SEND_BITS.RES0.PB22;
    TEST_BITS.OUT21 ON RCV_BITS.RES0.OUT21;
    TEST_BITS.IN22 ON SEND_BITS.RES0.IN22;
    TEST_BITS.OUT22 ON RCV_BITS.RES0.OUT22;
    TEST_BITS.PB31 ON SEND_BITS.RES0.PB31;
    TEST_BITS.IN31 ON SEND_BITS.RES0.IN31;
    TEST_BITS.OUT31 ON RCV_BITS.RES0.OUT31;
    TEST_BITS.PB32 ON SEND_BITS.RES0.PB32;
    TEST_BITS.IN32 ON SEND_BITS.RES0.IN32;
    TEST_BITS.OUT32 ON RCV_BITS.RES0.OUT32;
    TEST_INTS.PB1 ON SEND_INTS.RES0.PB1;
    TEST_INTS.IN1 ON SEND_INTS.RES0.IN1;
    TEST_INTS.PB2 ON SEND_INTS.RES0.PB2;
    TEST_INTS.IN2 ON SEND_INTS.RES0.IN2;
    TEST_INTS.PB3 ON SEND_INTS.RES0.PB3;
    TEST_INTS.IN3 ON SEND_INTS.RES0.IN3;
    TEST_INTS.PB4 ON SEND_INTS.RES0.PB4;
    TEST_INTS.IN4 ON SEND_INTS.RES0.IN4;
    TEST_INTS.OUT1 ON RCV_INTS.RES0.OUT1;
    TEST_INTS.OUT2 ON RCV_INTS.RES0.OUT2;
    TEST_INTS.OUT3 ON RCV_INTS.RES0.OUT3;
    TEST_INTS.OUT4 ON RCV_INTS.RES0.OUT4;
    TEST_UINTS.PB1 ON SEND_UINTS.RES0.PB1;
    TEST_UINTS.IN1 ON SEND_UINTS.RES0.IN1;
    TEST_UINTS.PB2 ON SEND_UINTS.RES0.PB2;
    TEST_UINTS.IN2 ON SEND_UINTS.RES0.IN2;
    TEST_UINTS.PB3 ON SEND_UINTS.RES0.PB3;
    TEST_UINTS.IN3 ON SEND_UINTS.RES0.IN3;
    TEST_UINTS.OUT1 ON RCV_UINTS.RES0.OUT1;
    TEST_UINTS.OUT2 ON RCV_UINTS.RES0.OUT2;
    TEST_UINTS.OUT3 ON RCV_UINTS.RES0.OUT3;
    TEST_REALS.PB1 ON SEND_REALS.RES0.PB1;
    TEST_REALS.IN1 ON SEND_REALS.RES0.IN1;
    TEST_REALS.PB2 ON SEND_REALS.RES0.PB2;
    TEST_REALS.IN2 ON SEND_REALS.RES0.IN2;
    TEST_REALS.OUT1 ON RCV_REALS.RES0.OUT1;
    TEST_REALS.OUT2 ON RCV_REALS.RES0.OUT2;
    TEST_TIMES.PB1 ON SEND_TIMES.RES0.PB1;
    TEST_TIMES.IN1 ON SEND_TIMES.RES0.IN1;
    TEST_TIMES.PB2 ON SEND_TIMES.RES0.PB2;
    TEST_TIMES.IN2 ON SEND_TIMES.RES0.IN2;
    TEST_TIMES.OUT1 ON RCV_TIMES.RES0.OUT1;
    TEST_TIMES.OUT2 ON RCV_TIMES.RES0.OUT2;
    TEST_STRINGS.PB1 ON SEND_STRINGS.RES0.PB1;
    TEST_STRINGS.IN1 ON SEND_STRINGS.RES0.IN1;
    TEST_STRINGS.PB2 ON SEND_STRINGS.RES0.PB2;
    TEST_STRINGS.IN2 ON SEND_STRINGS.RES0.IN2;
    TEST_STRINGS.OUT1 ON RCV_STRINGS.RES0.OUT1;
    TEST_STRINGS.OUT2 ON RCV_STRINGS.RES0.OUT2;
    TEST_ARRAY.PB1 ON SEND_ARRAY.RES0.PB1;
    TEST_ARRAY.IN1 ON SEND_ARRAY.RES0.PB1;
    TEST_ARRAY.OUT1 ON RCV_ARRAY.RES0.OUT1;
    TEST_COLOR.IN1 ON SEND_COLOR.RES0.IN1;
    TEST_COLOR.OUT1 ON RCV_COLOR.RES0.OUT1;
  END_MAPPINGS
END_SYSTEM
